FUNCTION_BLOCK Motor_Inversor (* Composite Function Block Type *)
  (* Standard: 61499-2 *)
  (* Version 0.0, 1/22/2026, Schneider Electric, template *)
  PACKAGE Hidryco.HidrycoLib;
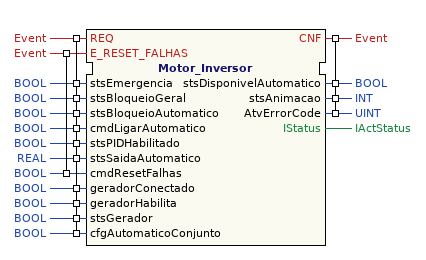
  EVENT_INPUT
    REQ WITH stsBloqueioGeral, stsBloqueioAutomatico, cmdLigarAutomatico, stsPIDHabilitado, stsSaidaAutomatico, geradorConectado, geradorHabilita, stsGerador, stsEmergencia, cfgAutomaticoConjunto; (* Normal Execution Request *)
    E_RESET_FALHAS WITH cmdResetFalhas;
  END_EVENT
  EVENT_OUTPUT
    CNF WITH stsDisponivelAutomatico, stsAnimacao, AtvErrorCode; (* Execution Confirmation *)
  END_EVENT
  VAR_INPUT
    stsEmergencia : BOOL;
    stsBloqueioGeral : BOOL;
    stsBloqueioAutomatico : BOOL;
    cmdLigarAutomatico : BOOL;
    stsPIDHabilitado : BOOL;
    stsSaidaAutomatico : REAL;
    cmdResetFalhas : BOOL;
    geradorConectado : BOOL;
    geradorHabilita : BOOL;
    stsGerador : BOOL;
    cfgAutomaticoConjunto : BOOL; (* 0 = Automatico Individual; 1 = Automatico em Conjunto *)
  END_VAR
  VAR_OUTPUT
    stsDisponivelAutomatico : BOOL;
    stsAnimacao : INT;
    AtvErrorCode : UINT; (* Current value(i) in the named variable array element *)
  END_VAR
  PLUGS
    IStatus : IActStatus;
  END_PLUGS
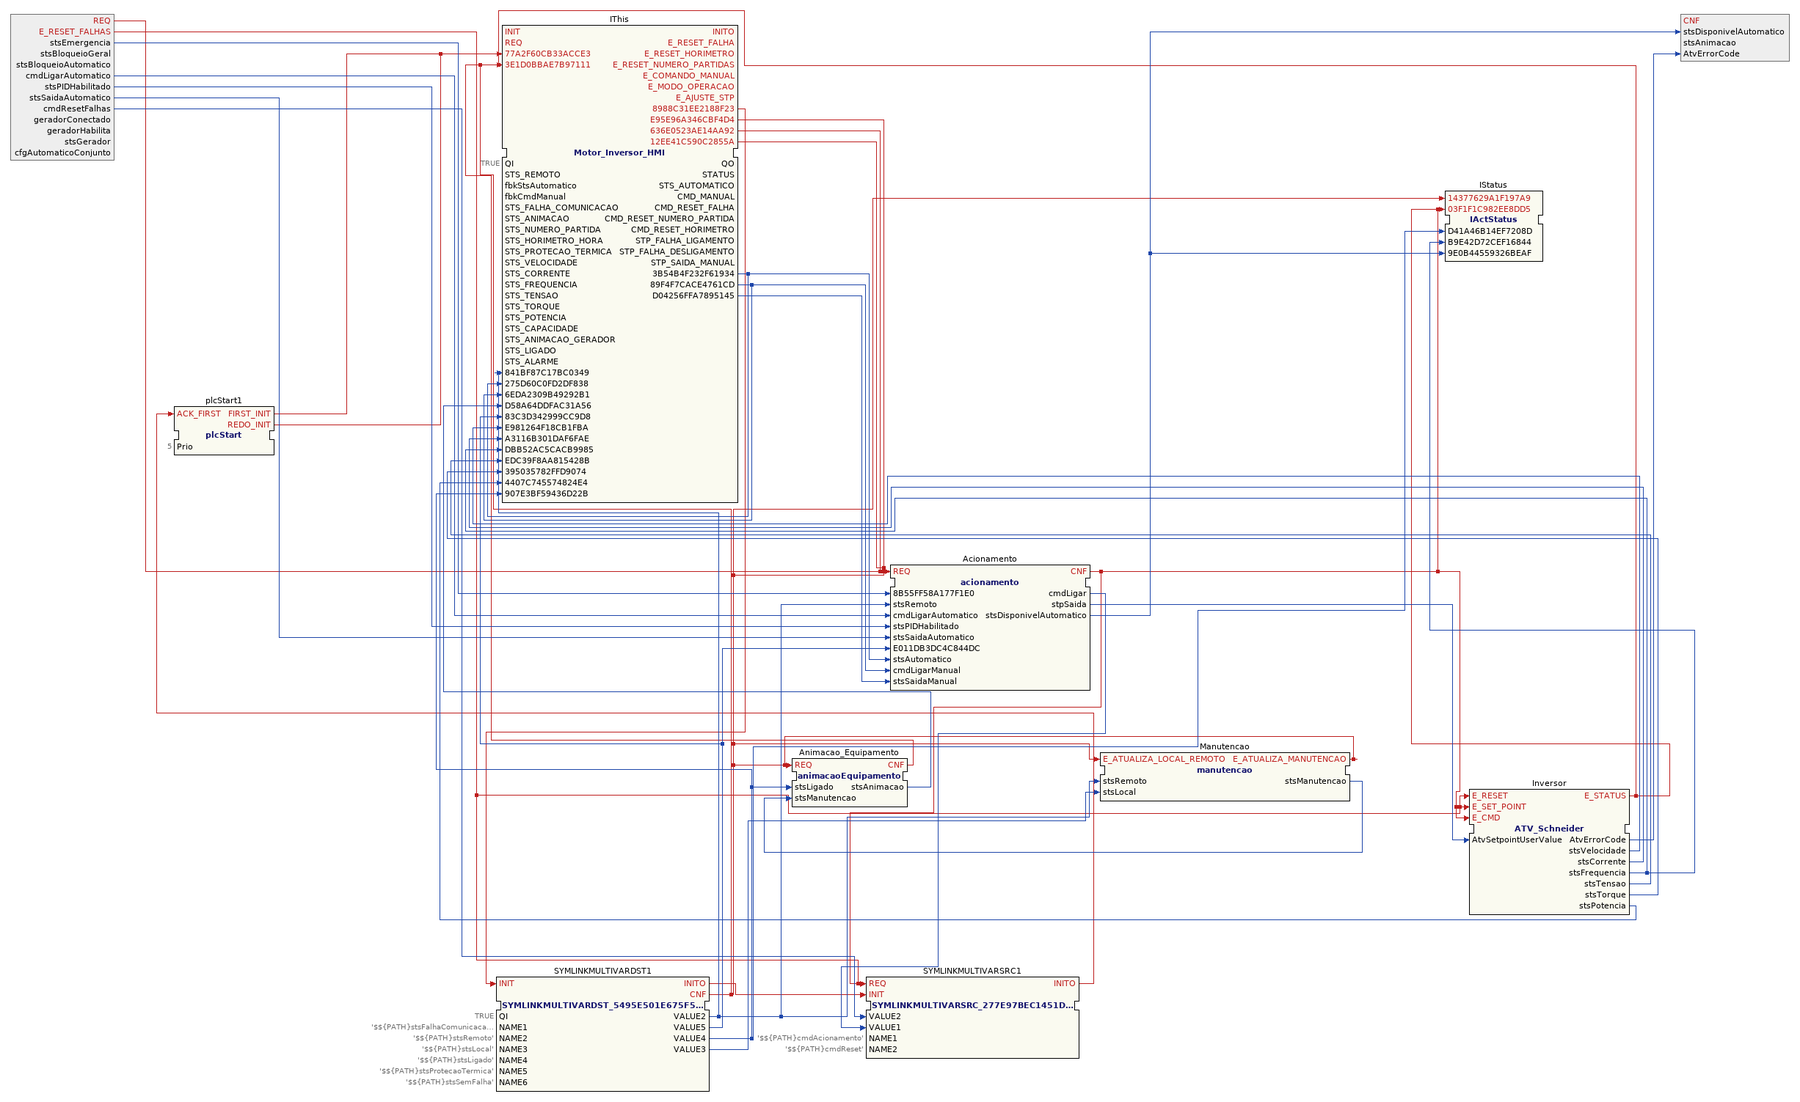
  (* 0 - INITIALIZATION *)
  (* 1 - FUNCTIONAL INPUT INTERFACE *)
  (* 6 - OT-IT INTERFACE *)
  (* 2 - FUNCTIONAL OUTPUT INTERFACE *)
  (* 3 - FIELD INTERFACE *)
  (* 4 - CHILDREN *)
  (* 5 - LOGICS *)
  (* 5.B - OPERATION MODE MANAGEMENT *)
  (* 5.A - FUNCTIONAL BEHAVIORS *)
  FBS
    IThis : Motor_Inversor_HMI(QI := TRUE);
    SYMLINKMULTIVARDST1 : SYMLINKMULTIVARDST_5495E501E675F500(QI := TRUE, NAME1 := '$${PATH}stsFalhaComunicacao', NAME2 := '$${PATH}stsRemoto', NAME3 := '$${PATH}stsLocal', NAME4 := '$${PATH}stsLigado', NAME5 := '$${PATH}stsProtecaoTermica', NAME6 := '$${PATH}stsSemFalha'); {SET_ATTRIBUTE(Configuration.GenericFBType.InterfaceParams, Runtime.System#I:=6;VALUE${I$}:BOOL,BOOL,BOOL,BOOL,BOOL,BOOL)}
    Inversor : ATV_Schneider;
    plcStart1 : plcStart(Prio := 5);
    SYMLINKMULTIVARSRC1 : SYMLINKMULTIVARSRC_277E97BEC1451D2C(NAME1 := '$${PATH}cmdAcionamento', NAME2 := '$${PATH}cmdReset'); {SET_ATTRIBUTE(Configuration.GenericFBType.InterfaceParams, Runtime.System#I:=2;VALUE${I$}:BOOL,BOOL)}
    Acionamento : acionamento;
    Animacao_Equipamento : animacaoEquipamento;
    Manutencao : manutencao;
  END_FBS
  EVENT_CONNECTIONS
    E_RESET_FALHAS TO Inversor.E_RESET;
    SYMLINKMULTIVARSRC1.INITO TO plcStart1.ACK_FIRST;
    E_RESET_FALHAS TO SYMLINKMULTIVARSRC1.REQ;
    SYMLINKMULTIVARDST1.INITO TO SYMLINKMULTIVARSRC1.INIT;
    REQ TO Acionamento.REQ;
    SYMLINKMULTIVARDST1.CNF TO Acionamento.REQ;
    Acionamento.CNF TO SYMLINKMULTIVARSRC1.REQ;
    Acionamento.CNF TO Inversor.E_SET_POINT;
    Acionamento.CNF TO Inversor.E_CMD;
    SYMLINKMULTIVARDST1.CNF TO Animacao_Equipamento.REQ;
    SYMLINKMULTIVARDST1.CNF TO Manutencao.E_ATUALIZA_LOCAL_REMOTO;
    Manutencao.E_ATUALIZA_MANUTENCAO TO Animacao_Equipamento.REQ;
    plcStart1.FIRST_INIT TO IThis.77A2F60CB33ACCE3;
    plcStart1.REDO_INIT TO IThis.77A2F60CB33ACCE3;
    Inversor.E_STATUS TO IThis.3E1D0BBAE7B97111;
    SYMLINKMULTIVARDST1.CNF TO IThis.3E1D0BBAE7B97111;
    Animacao_Equipamento.CNF TO IThis.3E1D0BBAE7B97111;
    IThis.8988C31EE2188F23 TO SYMLINKMULTIVARDST1.INIT;
    IThis.E95E96A346CBF4D4 TO Acionamento.REQ;
    IThis.636E0523AE14AA92 TO Acionamento.REQ;
    IThis.12EE41C590C2855A TO Acionamento.REQ;
    SYMLINKMULTIVARDST1.CNF TO IStatus.14377629A1F197A9;
    Inversor.E_STATUS TO IStatus.03F1F1C982EE8DD5;
    Acionamento.CNF TO IStatus.03F1F1C982EE8DD5;
  END_CONNECTIONS
  DATA_CONNECTIONS
    Inversor.AtvErrorCode TO AtvErrorCode;
    cmdResetFalhas TO SYMLINKMULTIVARSRC1.VALUE2;
    stsEmergencia TO Acionamento.8B55FF58A177F1E0;
    SYMLINKMULTIVARDST1.VALUE2 TO Acionamento.stsRemoto;
    cmdLigarAutomatico TO Acionamento.cmdLigarAutomatico;
    stsPIDHabilitado TO Acionamento.stsPIDHabilitado;
    stsSaidaAutomatico TO Acionamento.stsSaidaAutomatico;
    SYMLINKMULTIVARDST1.VALUE5 TO Acionamento.E011DB3DC4C844DC;
    Acionamento.cmdLigar TO SYMLINKMULTIVARSRC1.VALUE1;
    Acionamento.stpSaida TO Inversor.AtvSetpointUserValue;
    Acionamento.stsDisponivelAutomatico TO stsDisponivelAutomatico;
    SYMLINKMULTIVARDST1.VALUE4 TO Animacao_Equipamento.stsLigado;
    SYMLINKMULTIVARDST1.VALUE2 TO Manutencao.stsRemoto;
    SYMLINKMULTIVARDST1.VALUE3 TO Manutencao.stsLocal;
    Manutencao.stsManutencao TO Animacao_Equipamento.stsManutencao;
    SYMLINKMULTIVARDST1.VALUE2 TO IThis.841BF87C17BC0349;
    IThis.3B54B4F232F61934 TO IThis.275D60C0FD2DF838;
    IThis.89F4F7CACE4761CD TO IThis.6EDA2309B49292B1;
    Animacao_Equipamento.stsAnimacao TO IThis.D58A64DDFAC31A56;
    SYMLINKMULTIVARDST1.VALUE5 TO IThis.83C3D342999CC9D8;
    Inversor.stsVelocidade TO IThis.E981264F18CB1FBA;
    Inversor.stsCorrente TO IThis.A3116B301DAF6FAE;
    Inversor.stsFrequencia TO IThis.DBB52AC5CACB9985;
    Inversor.stsTensao TO IThis.EDC39F8AA815428B;
    Inversor.stsTorque TO IThis.395035782FFD9074;
    Inversor.stsPotencia TO IThis.4407C745574824E4;
    SYMLINKMULTIVARDST1.VALUE4 TO IThis.907E3BF59436D22B;
    IThis.3B54B4F232F61934 TO Acionamento.stsAutomatico;
    IThis.89F4F7CACE4761CD TO Acionamento.cmdLigarManual;
    IThis.D04256FFA7895145 TO Acionamento.stsSaidaManual;
    SYMLINKMULTIVARDST1.VALUE4 TO IStatus.D41A46B14EF7208D;
    Inversor.stsFrequencia TO IStatus.B9E42D72CEF16844;
    Acionamento.stsDisponivelAutomatico TO IStatus.9E0B44559326BEAF;
  END_CONNECTIONS
END_FUNCTION_BLOCK
